FUNCTION_BLOCK SDODatenMotorklemme1
VAR_INPUT
END_VAR
VAR_OUTPUT
	
	Motorklemme1Internaltemperature: SINT;
	Motorklemme1Steuerspannung: UINT;
	Motorklemme1Lastspannung: UINT;
	Motorklemme1Zykluszeit: UINT;
	Motorklemme1PWMFrequency: UINT;
		
END_VAR
VAR

	Internal_Temperature: FB_EcCoESdoRead;
	Control_Voltage: FB_EcCoESdoRead;
	Supply_Voltage: FB_EcCoESdoRead;
	Cycletime: FB_EcCoESdoRead;
	PWM_Frequency: FB_EcCoESdoRead;
	
	trigger: BOOL;
	TON_0: TON;
	TON_1: TON;
	ms: TIME;

END_VAR

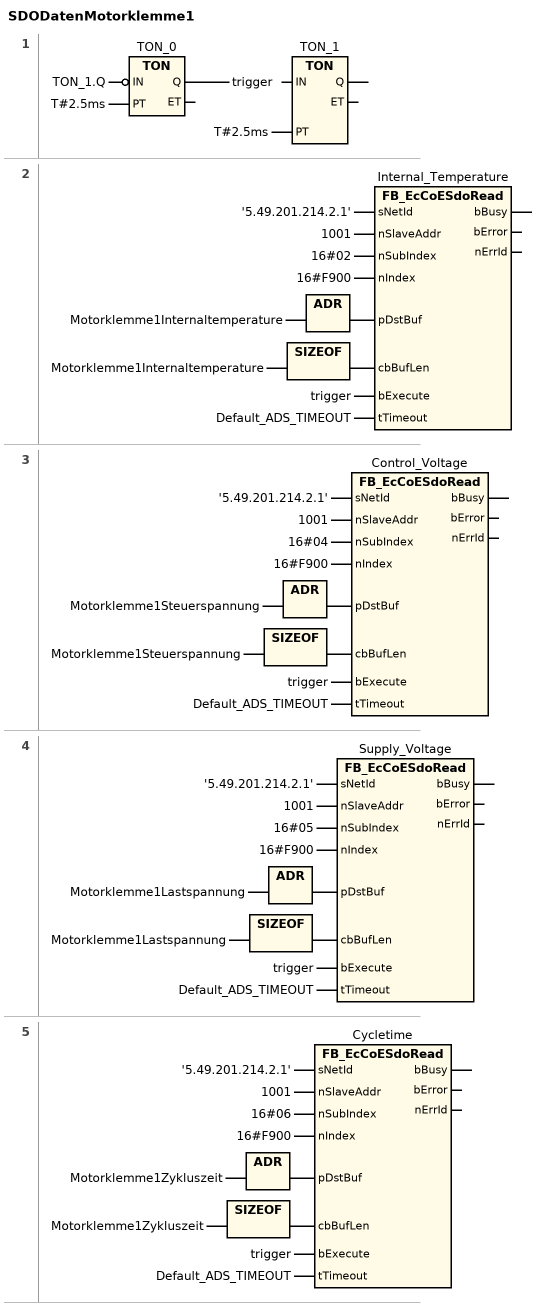
// NETWORK 1
TON_0(IN := NOT TON_1.Q, PT := T#2.5ms); // TON
trigger := TON_0.Q;
TON_1(IN := TON_0.Q, PT := T#2.5ms); // TON

// NETWORK 2
Internal_Temperature(
    sNetId := '5.49.201.214.2.1',
    nSlaveAddr := 1001,
    nSubIndex := 16#02,
    nIndex := 16#F900,
    pDstBuf := ADR(Motorklemme1Internaltemperature),
    cbBufLen := SIZEOF(Motorklemme1Internaltemperature),
    bExecute := trigger,
    tTimeout := Default_ADS_TIMEOUT); // FB_EcCoESdoRead

// NETWORK 3
Control_Voltage(
    sNetId := '5.49.201.214.2.1',
    nSlaveAddr := 1001,
    nSubIndex := 16#04,
    nIndex := 16#F900,
    pDstBuf := ADR(Motorklemme1Steuerspannung),
    cbBufLen := SIZEOF(Motorklemme1Steuerspannung),
    bExecute := trigger,
    tTimeout := Default_ADS_TIMEOUT); // FB_EcCoESdoRead

// NETWORK 4
Supply_Voltage(
    sNetId := '5.49.201.214.2.1',
    nSlaveAddr := 1001,
    nSubIndex := 16#05,
    nIndex := 16#F900,
    pDstBuf := ADR(Motorklemme1Lastspannung),
    cbBufLen := SIZEOF(Motorklemme1Lastspannung),
    bExecute := trigger,
    tTimeout := Default_ADS_TIMEOUT); // FB_EcCoESdoRead

// NETWORK 5
Cycletime(
    sNetId := '5.49.201.214.2.1',
    nSlaveAddr := 1001,
    nSubIndex := 16#06,
    nIndex := 16#F900,
    pDstBuf := ADR(Motorklemme1Zykluszeit),
    cbBufLen := SIZEOF(Motorklemme1Zykluszeit),
    bExecute := trigger,
    tTimeout := Default_ADS_TIMEOUT); // FB_EcCoESdoRead

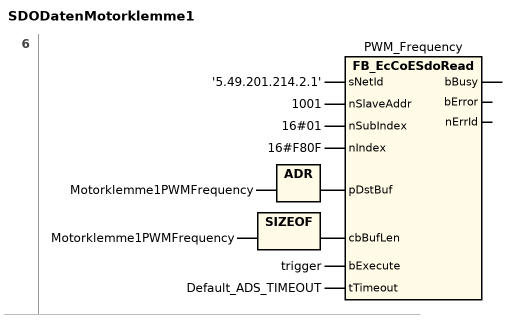
// NETWORK 6
PWM_Frequency(
    sNetId := '5.49.201.214.2.1',
    nSlaveAddr := 1001,
    nSubIndex := 16#01,
    nIndex := 16#F80F,
    pDstBuf := ADR(Motorklemme1PWMFrequency),
    cbBufLen := SIZEOF(Motorklemme1PWMFrequency),
    bExecute := trigger,
    tTimeout := Default_ADS_TIMEOUT); // FB_EcCoESdoRead

END_FUNCTION_BLOCK

(* stored: Version 1.1.0.1, ProductVersion 3.1.4020.12
   POU SDODatenMotorklemme1: Id {9f92255c-44a3-4130-a06c-2de7fbf9e0fd}, SpecialFunc None *)
